FUNCTION_BLOCK ABSTRACT FB_SystemContinous EXTENDS FB_ActorContinous
VAR_INPUT
END_VAR
VAR_OUTPUT
END_VAR
VAR
	{attribute 'OPC.UA.DA' := '1'}
	systemState : ST_SystemState;
END_VAR

METHOD PROTECTED ABSTRACT CheckError : BOOL
VAR_INPUT
END_VAR
VAR_OUTPUT
	bError : BOOL;
END_VAR
END_METHOD

METHOD PROTECTED MAIN : BOOL // Method that calls all needed function block methods
VAR_INPUT
END_VAR
SUPER^.MAIN();
SystemFlowControl();
END_METHOD

METHOD PROTECTED ABSTRACT Operational : BOOL
VAR_INPUT
END_VAR
VAR_OUTPUT
	bSwitchToWorking : BOOL := FALSE;
END_VAR
END_METHOD

METHOD PROTECTED ABSTRACT RampDown : BOOL
VAR_INPUT
END_VAR
VAR_OUTPUT
	bRampDownFinished : BOOL := FALSE;
END_VAR
END_METHOD

METHOD PROTECTED ABSTRACT RampUp : BOOL
VAR_INPUT
END_VAR
VAR_OUTPUT
	bRampUpFinished : BOOL := FALSE;
END_VAR
END_METHOD

METHOD PROTECTED ABSTRACT  SetSetPointLimits : BOOL
VAR_INPUT
END_VAR
END_METHOD

METHOD SystemFlowControl : INT
VAR_INPUT
END_VAR
VAR_INST
	nState : E_SystemOperatingState := E_SystemOperatingState.standby; //actual state number
	bSwitchState : BOOL := FALSE;
	bSystemError : BOOL := FALSE;
END_VAR
CheckError(bError => bSystemError);
systemState.bError := bSystemError;

IF NOT bSystemError THEN
	CASE nState OF
		E_SystemOperatingState.standby:
			systemState.sOperatingState := 'standby';
			bSwitchState := FALSE;
			//if turned on switch to ramp-up
			IF(bSetStatusOn) THEN
				nState := E_SystemOperatingState.rampUp;
			END_IF
		E_SystemOperatingState.rampUp:
			systemState.sOperatingState := 'ramp-up';
			RampUp(bRampUpFinished => bSwitchState);
			//if turned off switch to ramp-down
			IF(NOT bSetStatusOn) THEN
				nState := E_SystemOperatingState.rampDown;
			//if ramp-up finished switch to operational
			ELSIF(bSwitchState) THEN
				nState := E_SystemOperatingState.operational;
			END_IF
		E_SystemOperatingState.operational:
			systemState.sOperatingState := 'operational';
			Operational(bSwitchToWorking => bSwitchState);
			//if turned off switch to ramp-down
			IF(NOT bSetStatusOn) THEN
				nState := E_SystemOperatingState.rampDown;
			//switch to working if desired
			ELSIF(bSwitchState) THEN
				nState := E_SystemOperatingState.working;
			END_IF
		E_SystemOperatingState.working:
			systemState.sOperatingState := 'working';
			Working(bSwitchToOperational => bSwitchState);
			//if turned off switch to ramp-down
			IF(NOT bSetStatusOn) THEN
				nState := E_SystemOperatingState.rampDown;
			//switch to operational if desired
			ELSIF(bSwitchState) THEN
				nState := E_SystemOperatingState.operational;
			END_IF
		E_SystemOperatingState.rampDown:
			systemState.sOperatingState := 'ramp-down';
			RampDown(bRampDownFinished => bSwitchState);
			//if turned on switch to ramp-up
			IF(bSetStatusOn) THEN
				nState := E_SystemOperatingState.rampUp;
			//if ramp-down finished switch to standby
			ELSIF(bSwitchState) THEN
				nState := E_SystemOperatingState.standby;
			END_IF
	END_CASE
ELSE
	RampDown(bRampDownFinished => bSwitchState);
	IF bSwitchState THEN
		systemState.sOperatingState := 'standby';
		nState := E_SystemOperatingState.standby;
	ELSE
		systemState.sOperatingState := 'ramp-down';	
		nState := E_SystemOperatingState.rampDown;		
	END_IF
	
END_IF
systemState.nOperatingState := nState;
END_METHOD

METHOD PROTECTED ABSTRACT Working : BOOL
VAR_INPUT
END_VAR
VAR_OUTPUT
	bSwitchToOperational : BOOL := FALSE;
END_VAR
END_METHOD

END_FUNCTION_BLOCK

(* stored: Version 1.1.0.1, ProductVersion 3.1.4024.9
   POU FB_SystemContinous: Id {96d5c5c8-8c8e-4fc0-9cb9-dd455bc0dccf}, SpecialFunc None
   Method CheckError: Id {ad935b5d-159a-45d8-a497-f9d6421f009b}
   Method MAIN: Id {0f6296ee-45f5-4e45-b70e-a6b0f33b8461}
   Method Operational: Id {2598fbd1-9bc6-46f7-b45a-1192dd4e31bf}
   Method RampDown: Id {c456b4e1-b9b4-4165-a480-69fcb8d85911}
   Method RampUp: Id {90e484f3-4a54-4088-a19e-e3315ad62ded}
   Method SetSetPointLimits: Id {76638cd5-20cb-42ab-afc6-a5afa22b29a7}
   Method SystemFlowControl: Id {6217cbf4-0afa-43b2-8f55-e14926bb4551}
   Method Working: Id {16283899-5654-440c-b82d-86196b3a2bb6} *)
